{attribute addProperty BoxType "AT2050-0500-0017"}
{attribute addProperty Id "A_0096_AT2025_5250_0017_AT2025_5250AT2025_3DCFC8D064080"}
{attribute addProperty CRC "1745998061"}
{attribute addProperty SizeInBites "640"}
{attribute addProperty SizeInBytes "80"}
TYPE A_0048_AT2050_0500_0017_6811D0ED EXTENDS AT2050_9506A482 :
STRUCT
	{attribute addProperty Name "A_0096_AT2025_5250_0017_AT2025_5250"}
	A_0096_AT2025_5250_0017_AT2025_5250 : AT2025_3DCFC8D0;
END_STRUCT
END_TYPE

(* stored: Version 1.2.0.0, ProductVersion 3.1.4024.9
   DUT A_0048_AT2050_0500_0017_6811D0ED: Id {a90d8f36-1662-4838-8e82-903f11f29060} *)
